Fanuc KAREL source: INV.kl

PROGRAM T
%NOLOCKGROUP
VAR
 v0 : POSITION
 res : POSITION
BEGIN
 res = INV(v0)
END T
